{attribute addProperty BoxType "EP9224-0037-0017"}
{attribute addProperty Id "Device_StatusAT %I*Device_Status_3F5AD3531621Current_UsAT %I*INT16217Current_UpAT %I*INT16218Voltage_UsAT %I*INT16219Voltage_UpAT %I*INT16220TemperatureAT %I*INT16221"}
{attribute addProperty CRC "3257998778"}
{attribute addProperty SizeInBites "96"}
{attribute addProperty SizeInBytes "12"}
TYPE DPO_Inputs_Device_C2311DBA :
STRUCT
	{attribute addProperty Name "Device_Status"}
	Device_Status AT %I* : Device_Status_3F5AD353;
	{attribute addProperty Name "Current_Us"}
	Current_Us AT %I* : INT;
	{attribute addProperty Name "Current_Up"}
	Current_Up AT %I* : INT;
	{attribute addProperty Name "Voltage_Us"}
	Voltage_Us AT %I* : INT;
	{attribute addProperty Name "Voltage_Up"}
	Voltage_Up AT %I* : INT;
	{attribute addProperty Name "Temperature"}
	Temperature AT %I* : INT;
END_STRUCT
END_TYPE

(* stored: Version 1.2.0.0, ProductVersion 3.1.4024.9
   DUT DPO_Inputs_Device_C2311DBA: Id {d71e21bc-69ed-4214-bb7b-04ccd97e6eae} *)
